PROGRAM MAIN
VAR
END_VAR

LLD();

END_PROGRAM

(* stored: Version 1.1.0.1, ProductVersion 3.1.4024.12
   POU MAIN: Id {068c917d-6832-4147-af64-3966d0d4b503}, SpecialFunc None *)
